ABB RobotStudio station: practica3_EstacionDePartida_1.rspag

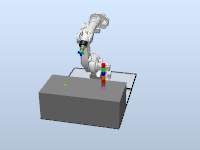
--- station ---
Station practica3_EstacionDePartida_1 (saved by RobotStudio 20.4.9280.0)
Controller Sistema6
  mechanical unit ROB_1: IRB6640_180_255__04, 6 joints, base frame (0, 0, 0) mm
Layout (positions relative to the parent item):
  - Ventosa [mechanism] at (1619.04, 42.44, 1910.18) mm, rotated rx -180 ry 54.91 rz -180 deg
      TCP Ventosa at (0, 0, 200) mm
      links: PiezaVentosa
  - IRB6640_180_255__04 [mechanism, from Robots\IRB6640_180_255_G_04.rslib] at (0, 0, 0) mm; joint values [0.0291, -0.0105, 0.0365, -0.043, 0.5871, 0.0526] (rad or m)
  - MesaTrabajoParteIzq [part]
  - MesaTrabajoParteDer [part]
  - CI_VentosaVacuostato [smart component]
      signals: DI ActivaVentosa, DO Vacuostato
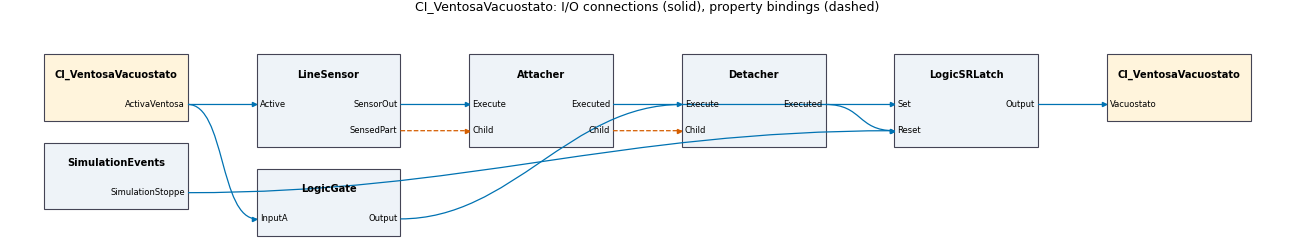
      connections:
        CI_VentosaVacuostato.ActivaVentosa -> LineSensor.Active
        LineSensor.SensorOut -> Attacher.Execute
        Attacher.Executed -> LogicSRLatch.Set
        LogicSRLatch.Output -> CI_VentosaVacuostato.Vacuostato
        Detacher.Executed -> LogicSRLatch.Reset
        SimulationEvents.SimulationStopped -> LogicSRLatch.Reset
        CI_VentosaVacuostato.ActivaVentosa -> LogicGate.InputA
        LogicGate.Output -> Detacher.Execute
        LineSensor.SensedPart => Attacher.Child
        Attacher.Child => Detacher.Child
    - LineSensor [smart component, from Components\LineSensor.rslib] at (1782.69, 42.44, 1795.2) mm, rotated rx -180 ry 54.91 rz -180 deg
        properties: Start=[0 0 -0.002]; End=[0 0 0.02]; Radius=0.002; SensedPart=(none); SensedPoint=[1.78268933105469 0.0424414672851562 1.7952001953125]
      - _sensorPart_ [part]
    - SimulationEvents [smart component, from Components\SimulationEvents.rslib]
    - LogicSRLatch [smart component, from Components\LogicSRLatch.rslib]
    - Attacher [smart component, from Components\Attacher.rslib]
        properties: Parent=Ventosa; Flange=0; Child=(none); Mount=false; Offset=[0 0 0]; Orientation=[0 0 0]
    - Detacher [smart component, from Components\Detacher.rslib]
        properties: Child=(none); KeepPosition=true
    - LogicGate [smart component, from Components\LogicGate.rslib]
        properties: Operator=NOT; Delay=0.1
  - Pieza_8 [part]
  - Pieza_15 [part]
  - Pieza_16 [part]
  - Pieza_17 [part]
  - Pieza_18 [part]
  - Pieza_19 [part]
  - Pieza_20 [part]
Attachment: LineSensor is attached to Ventosa / PiezaVentosa
Attachment: Ventosa is attached to IRB6640_180_255__04 / Link6
Station logic (signal -> signal, property => property):
  CI_VentosaVacuostato.Vacuostato -> Sistema6.ED_PiezaCogida
  Sistema6.SD_ActivaVentosa -> CI_VentosaVacuostato.ActivaVentosa

--- Backups/Sistema6/RAPID/TASK1/PROGMOD/CalibData.mod ---
MODULE CalibData
	PERS tooldata Ventosa:=[TRUE,[[0,0,200],[1,0,0,0]],[1,[0,0,125],[1,0,0,0],0.002,0.002,0.0013]];
ENDMODULE

--- Backups/Sistema6/RAPID/TASK1/PROGMOD/Module1.mod ---
MODULE Module1
	CONST robtarget pReposo:=[[1808.910161514,0,1855],[0.5,0,0.866025404,0],[0,0,0,0],[9E+09,9E+09,9E+09,9E+09,9E+09,9E+09]];
	CONST robtarget pBaseTorre1:=[[1500,500,750],[0,0,1,0],[0,0,0,0],[9E+09,9E+09,9E+09,9E+09,9E+09,9E+09]];
    CONST robtarget pBaseTorre2:=[[1500,-500,750],[0,0,1,0],[0,0,0,0],[9E+09,9E+09,9E+09,9E+09,9E+09,9E+09]];

    CONST num diametro := 100;
    CONST num altura := 100;



PROC main()
    ! Movemos la primera torre de 7 piezas 2 veces el diametro de la pieza
    MueveTorre pBaseTorre1, pBaseTorre2, 7, 5;

ENDPROC

PROC MueveTorre(robtarget pOrigen,robtarget pDestino, num nPiezas, num desplazamiento)
   !Array donde vamos a guardar todos los puntos para usarlos en un bucle FOR
   VAR robtarget tabPos{3}; !Punto inicial, intermedio, y final
   VAR robtarget pIntermedio;
   VAR robtarget pAproxMonton1;
   VAR robtarget pAproxMonton2;
   VAR robtarget pMonton1;
   VAR robtarget pMonton2;

   !Creamos el punto intermedio con la altura inicial
   pIntermedio := Offs (pOrigen, 0, diametro * desplazamiento * (-1), altura);

   !Añadimos los 3 puntos a la tabla
   tabPos{1} := pOrigen;
   tabPos{2} := pIntermedio;
   tabPos{3} := pDestino;

   !Creamos el bucle FOR
   FOR i FROM 1 TO 2 DO !Recorreremos el bucle primero con los puntos i e i+1 y despues con i+1 e i+2

   !Definimos los puntos iniciales de los dos montones
   pMonton1 := Offs (tabPos{i}, 0, 0, altura * nPiezas);
   pMonton2 := Offs (tabPos{i+1}, 0, 0, altura);

    !Creamos los 3 puntos de aproximación
   pAproxMonton1 := Offs (tabPos{i}, 0, 0, (altura * nPiezas) + altura);
   pAproxmonton2 := Offs (tabPos{i+1}, 0, 0, (altura * nPiezas) + altura);

    FOR nPiezas2 FROM 1 TO nPiezas DO !Bucle para el número de piezas

        !Movemos el brazo a la posición de aproximación del monton 1
        MoveL pAproxMonton1, v2000, fine, Ventosa\WObj:=wobj0;

        !Cogemos la pieza del monton 1
        MoveLDO pMonton1, v2000, fine, Ventosa\WObj:=wobj0, SD_ActivaVentosa, 1;
        WaitDI ED_PiezaCogida, 1; !Esperamos a que PiezaCogida esté a 1
        MoveL pAproxMonton1, v2000, fine, Ventosa\WObj:=wobj0;

        !Movemos el brazo a la posicion de aproximación del monton 2
        MoveL pAproxmonton2, v2000, fine, Ventosa\WObj:=wobj0;

        !Ponemos la pueza en el montón 2
        MoveLDO pMonton2, v2000, fine, Ventosa\WObj:=wobj0, SD_ActivaVentosa, 0;
        WaitDI ED_PiezaCogida, 0; !Esperamos a que PiezaCogida esté a 1
        MoveL pAproxmonton2, v2000, fine, Ventosa\WObj:=wobj0;

        !Calculamos los nuevos puntos de cada montón
        pMonton1 := Offs (pMonton1, 0, 0, - altura);
        pMonton2 := Offs (pMonton2, 0, 0, altura);

    ENDFOR
   ENDFOR



ENDPROC

ENDMODULE

--- Backups/Sistema6/RAPID/TASK1/SYSMOD/LINKEDM.sys ---
%%%
  VERSION:1
  LANGUAGE:ENGLISH
%%%

MODULE LINKEDM (SYSMODULE)

! FOLLOWER
!     Name of electronically linked follower axis used by operator at teach pendent.
      PERS string l_f_axis_name{5}       :=  ["",  "", "", "", ""];

!     Name of the mechanical unit for follower axis.
      PERS string l_f_mecunt_n{5}  :=  ["", "", "", "", ""];

!     Linked follower axis number in the mechanical unit (first axis in mech. unit is number 1).
      PERS num l_f_axis_no{5}      :=  [0,          0,   0,  0,  0];

! MASTER
!     Name of the mechanical unit for linked master axis.
      PERS string l_m_mecunt_n{5} :=  ["", "", "", "", ""];

!     Linked master axis number in the mechanical unit (first axis in mech. unit is number 1).
!     See axis number table in documentation for different master mechanical units.
      PERS num l_m_axis_no{5}     :=  [0,  0,  0,  0,  0];

! POSITION OFFSET
!     The increase of the allowed offset position between the master and follower
!     positions, used when starting AUTO mode. As soon as the offset is decreased
!     the old configurated parameter is used.
!     Example: 3 => the configurated value of allowed offset is increased 3 times.
      PERS num offset_ratio{5}       :=  [10,  10,   10,  10,  10];

! SPEED RATIO
!     Speed_ratio used in AUTO and JOG modes [ very_slow   slow    normal    fast]
!     Value 1 = max allowed manual speed.
      CONST num speed_ratio {20}      := [0.01, 0.01, 0.01, 0.01, 0.01,
                                          0.05, 0.05, 0.05, 0.05, 0.05,
                                          0.20, 0.20, 0.20, 0.20, 0.20,
                                          1.00, 1.00, 1.00, 1.00, 1.00];

! STEP SIZE
!     Displacement position used in JOG mode for each activation of positive or
!     negative movement.                  [very_short    short   normal   long]
!     Unit degees or meter.
      CONST num displacement {20}     := [0.001, 0.001, 0.001, 0.001, 0.001,
                                          0.005, 0.005, 0.005, 0.005, 0.005,
                                          0.020, 0.020, 0.020, 0.020, 0.020,
                                          0.100, 0.100, 0.100, 0.100, 0.100];


!-------------------------------------------------------------
 PROC Linked_m ()
      Linked_m_exe ;
 ENDPROC
ENDMODULE

--- Backups/Sistema6/SYSPAR/EIO.cfg ---
EIO:CFG_1.0:6:1::
#
INDUSTRIAL_NETWORK:

      -Name "DeviceNet" -Label "DeviceNet Master/Slave Network" -Address "2"
#
DEVICENET_DEVICE:

      -Name "MiDeviceNet" -Label "MiDeviceNet"
#
DEVICENET_INTERNAL_DEVICE:

      -Name "DN_Internal_Device" -VendorName "ABB Robotics"\
      -ProductName "DeviceNet Internal Slave Device"
#
EIO_SIGNAL:

      -Name "ED_PiezaCogida" -SignalType "DI" -Device "MiDeviceNet"\
      -Label "ED_PiezaCogida" -DeviceMap "0" -Access "All"

      -Name "SD_ActivaVentosa" -SignalType "DO" -Device "MiDeviceNet"\
      -Label "SD_ActivaVentosa" -DeviceMap "0" -Access "All"
